
FUNCTION CB_shl_sint : INT


TITLE = ' shift on bit string '
VERSION : '1.0'
AUTHOR  : CB
NAME    : shlSint
FAMILY  : TNI

VAR_INPUT
    IN : INT;
    N : INT;
END_VAR

BEGIN

    CB_shl_sint := BYTE_TO_INT(SHL(IN := INT_TO_BYTE(IN), N := N));

END_FUNCTION
